VAR_GLOBAL
	sDatastring: STRING(500);
	
	Moteeui			: STRING;
	Appeui			: STRING;
	UserData		: ST_UserData;
	PayloadDecoded	: STRING;

	PayloadLength	: DINT;
	PayloadData		: ARRAY[1..100] OF BYTE;
	NullByte		: BYTE := 0;

END_VAR

(* stored: Version 1.1.0.1, ProductVersion 3.1.4022.7
   GVL GVL_1: Id {385ba8bf-824b-4bcb-9d7a-e08cfee83de9} *)
